# EPICS autosave request: iocBoot/sioc-esb-bkh17/bkh17.req
file ../bkhDigiO.req P=$(P),MOD=2114-$(M),N=1
file ../bkhDigiO.req P=$(P),MOD=2114-$(M),N=2
file ../bkhDigiO.req P=$(P),MOD=2114-$(M),N=3
file ../bkhDigiO.req P=$(P),MOD=2114-$(M),N=4
file ../bkhDigiO.req P=$(P),MOD=2114-$(M),N=5
file ../bkhDigiO.req P=$(P),MOD=2114-$(M),N=6
file ../bkhDigiO.req P=$(P),MOD=2114-$(M),N=7
file ../bkhDigiO.req P=$(P),MOD=2114-$(M),N=8

file ../bkhDigiO.req P=$(P),MOD=2124-$(M),N=1
file ../bkhDigiO.req P=$(P),MOD=2124-$(M),N=2
file ../bkhDigiO.req P=$(P),MOD=2124-$(M),N=3
file ../bkhDigiO.req P=$(P),MOD=2124-$(M),N=4
file ../bkhDigiO.req P=$(P),MOD=2124-$(M),N=5
file ../bkhDigiO.req P=$(P),MOD=2124-$(M),N=6
file ../bkhDigiO.req P=$(P),MOD=2124-$(M),N=7
file ../bkhDigiO.req P=$(P),MOD=2124-$(M),N=8

file ../bkhDigiI.req P=$(P),MOD=1124-$(M),N=1
file ../bkhDigiI.req P=$(P),MOD=1124-$(M),N=2
file ../bkhDigiI.req P=$(P),MOD=1124-$(M),N=3
file ../bkhDigiI.req P=$(P),MOD=1124-$(M),N=4

file ../bkhDigiI.req P=$(P),MOD=1104-$(M),N=1
file ../bkhDigiI.req P=$(P),MOD=1104-$(M),N=2
file ../bkhDigiI.req P=$(P),MOD=1104-$(M),N=3
file ../bkhDigiI.req P=$(P),MOD=1104-$(M),N=4
